// TIA Portal V16 export
// export: Created 2021-05-24T12:27:50.3765548Z, ExportSetting WithDefaults, DisplayName Totally Integrated Automation Portal, DisplayVersion V16 Update 3, DisplayName TIA Portal Version Control Interface, DisplayVersion V16 Update 2, DisplayName TIA Portal Openness, DisplayVersion V16 Update 3, DisplayName STEP 7 Professional, DisplayVersion V16 Update 3, DisplayName STEP 7 Safety, DisplayVersion V16, DisplayName WinCC Professional, DisplayVersion V16 Update 3
DATA_BLOCK "DB38151_Dy_SubTimeEventRTC"   // DB38151
TITLE = Dynamic DB — Subroutine - Event Timer Using RTC
{ S7_Optimized_Access := 'TRUE' }
AUTHOR : M_Gledhill
FAMILY : Subroutine
NAME : Dy_SubTimeEventRTC
VERSION : 1.0
// PRACTICAL SERIES AUTOMATION LIBRARY (PAL)   —   COPYRIGHT 2020 – M. GLEDHILL (MIT LICENCE)
//                   ———— ◆ ————
//  FOR DETAILED DOCUMENTATION — SELECT THE BLOCK IN THE PROJECT TREE AND PRESS SHIFT + F1
//  FULL ONLINE DOCUMENTATION IS AVAILABLE AT: https://practicalseries.com/2001-pal/index.html
// stored: AutoNumber false, DBAccessibleFromOPCUA true, IsOnlyStoredInLoadMemory false, IsRetainMemResEnabled false, IsWriteProtectedInAS false, MemoryReserve 100
   VAR
      _DB_Header { ExternalAccessible := 'False'; ExternalVisible := 'False'; ExternalWritable := 'False'} : Array[0..79] of Bool;   // SUBROUTINE EVENT TIMER USING RTC
      __________0000_0 { ExternalWritable := 'False'} : Bool := false;
      __________0000_1 { ExternalWritable := 'False'} : Bool := false;   // ▀▀▀▀ DB CURRENT REVISION
      revInfo { ExternalWritable := 'False'} : "UT01000_St_SysRevision";
      __________0010_0 { ExternalAccessible := 'False'; ExternalVisible := 'False'; ExternalWritable := 'False'} : Bool := false;
      __________0010_1 { ExternalAccessible := 'False'; ExternalVisible := 'False'; ExternalWritable := 'False'} : Bool := false;   // ▀▀▀▀ SYSTEM EVENT TIMER
      FC18151_Event { ExternalWritable := 'False'} : "UT38151_Dy_SubTimeEventRTC";   // Event timer — 1 Day
      FC02001_AlmH_OnTime { ExternalWritable := 'False'; S7_SetPoint := 'True'} : "UT38151_Dy_SubTimeEventRTC";   // FC02001 Test — Alarm High On Time
      FC02001_AlmH_OffTime { ExternalWritable := 'False'; S7_SetPoint := 'True'} : "UT38151_Dy_SubTimeEventRTC";   // FC02001 Test — Alarm High Off Time
      FC02001_AlmL_OnTime { ExternalWritable := 'False'; S7_SetPoint := 'True'} : "UT38151_Dy_SubTimeEventRTC";   // FC02001 Test — Alarm Low On Time
      FC02001_AlmL_OffTime { ExternalWritable := 'False'; S7_SetPoint := 'True'} : "UT38151_Dy_SubTimeEventRTC";   // FC02001 Test — Alarm Low Off Time
      FC02001_WrnH_OnTime { ExternalWritable := 'False'; S7_SetPoint := 'True'} : "UT38151_Dy_SubTimeEventRTC";   // FC02001 Test — Warning High On Time
      FC02001_WrnH_OffTime { ExternalWritable := 'False'; S7_SetPoint := 'True'} : "UT38151_Dy_SubTimeEventRTC";   // FC02001 Test — Warning High Off Time
      FC02001_WrnL_OnTime { ExternalWritable := 'False'; S7_SetPoint := 'True'} : "UT38151_Dy_SubTimeEventRTC";   // FC02001 Test — Warning Low On Time
      FC02001_WrnL_OffTime { ExternalWritable := 'False'; S7_SetPoint := 'True'} : "UT38151_Dy_SubTimeEventRTC";   // FC02001 Test — Warning Low Off Time
   END_VAR
BEGIN
   // _DB_Header[0] : ▀▀▀▀▀▀▀▀▀▀▀▀▀▀▀▀▀▀▀▀▀▀▀▀▀▀▀▀▀▀▀▀▀▀▀▀▀▀▀▀▀▀▀▀
   // _DB_Header[2] : TITLE: SUBROUTINE EVENT TIMER USING RTC
   // _DB_Header[4] : ▄▄▄▄▄▄▄▄▄▄▄▄▄▄▄▄▄▄▄▄▄▄▄▄▄▄▄▄▄▄▄▄▄▄▄▄▄▄▄▄▄▄▄▄
   // _DB_Header[5] : TYPE: DYNAMIC
   // _DB_Header[6] : ▀▀▀▀▀▀▀▀▀▀▀▀▀▀▀▀▀▀▀▀▀▀▀▀▀▀▀▀▀▀▀▀▀▀▀▀▀▀▀▀▀▀▀▀
   // _DB_Header[8] : This is the dynamic data block associated with the event timing subroutine block
   // _DB_Header[10] : FC18151_SubTimeEventRTC
   // _DB_Header[12] : The dynamic data holds the event start time, end time and duration
   // _DB_Header[14] : Each event is given the user data type:
   // _DB_Header[15] : UT18151_Dy_SubTimeEventRTC
   // _DB_Header[19] : ━━━ ⬙⬙⬙⬙⬙⬙ ━━━
   // _DB_Header[21] : ▄▄▄▄▄▄▄▄▄▄▄▄▄▄▄▄▄▄▄▄▄▄▄▄▄▄▄▄▄▄▄▄▄▄▄▄▄▄▄▄▄▄▄▄
   // _DB_Header[22] : MODIFICATION HISTORY
   // _DB_Header[24] : This is a summary of the recent software modifications made to this block (most recent at top)
   // _DB_Header[26] : ―――――――――――――――――――――――――――――――――――――――――――
   // _DB_Header[27] : DATE REVISION MASTER BRANCH DEV
   // _DB_Header[28] : (nnn.amm) COMMIT TAG (Base ---> Merge) BRANCH Author
   // _DB_Header[29] : ———————————————————————————————————————————
   // _DB_Header[30] : 2021.02.19 001.000 D0003 D0002 D0003 None M. Gledhill
   // _DB_Header[31] : FC18151 — RELEASED FOR USE
   // _DB_Header[32] : Merge back to master branch
   // _DB_Header[34] : 2021.02.19 001.000 D0002A-001.000 D0002 N/A D0002A M. Gledhill
   // _DB_Header[35] : FC18151 — Post test RELEASED FOR USE
   // _DB_Header[37] : 2021.02.18 000.801 D0002A-000.801 D0002 N/A D0002A M. Gledhill
   // _DB_Header[38] : FC18151 Migration to VCS — Released for test
   // _DB_Header[39] : ———————————————————————————————————————————
   // _DB_Header[40] : Where: nnn = Major revision
   // _DB_Header[41] : a = Type (1-7 Development, 8 Proving, 9 Qualification, 0 Release)
   // _DB_Header[42] : mm = Minor revision (must be 00 if a = 0)
   // _DB_Header[43] : Block properties version number should be set to nn.a (only one decimal place)
   // _DB_Header[45] : ██████████████ █ █ █ █ END █ █ █ █ ██████████████
   revInfo.REV_BLOCK := 'DB38151';
   revInfo.REV_NUMBER := '001.000';
   revInfo.REV_DATE := '2021-02-19';
   revInfo.REV_AUTHOR := 'M. Gledhill';
END_DATA_BLOCK
